// TIA Portal V18 export
// export: Created 2026-06-08T17:17:40.8310714Z, ExportSetting WithDefaults, DisplayName Totally Integrated Automation Portal, DisplayVersion V18, DisplayName TIA Portal Openness, DisplayVersion V18, DisplayName TIA Portal Version Control Interface, DisplayVersion V18, DisplayName STEP 7 Professional, DisplayVersion V18, DisplayName STEP 7 Safety, DisplayVersion V18, DisplayName WinCC Professional, DisplayVersion V18
ORGANIZATION_BLOCK "Main"   // OB1, LAD, ProgramCycle
TITLE = "Main Program Sweep (Cycle)"
{ S7_Optimized_Access := 'TRUE' }
VERSION : 0.1
// stored: AutoNumber true, IsIECCheckEnabled false, SetENOAutomatically false
BEGIN

REGION Network 1
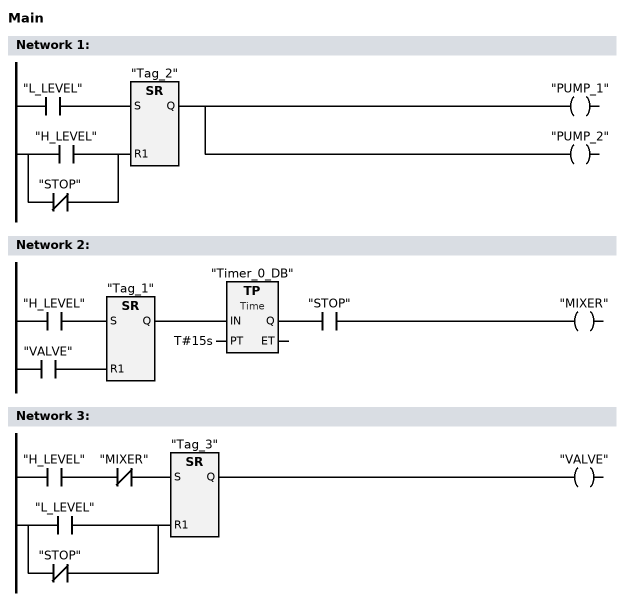
   RUNG wire#powerrail
      Contact( "L_LEVEL" )
      S_SR(operand := "Tag_2", r1 := wire#w1)
      wire#w2
      Coil( "PUMP_1" )
   END_RUNG
   RUNG wire#powerrail
      Contact( "H_LEVEL" )
   END_RUNG wire#w1
   RUNG wire#powerrail
      I_Contact( "STOP" )
   END_RUNG wire#w1
   RUNG wire#w2
      Coil( "PUMP_2" )
   END_RUNG
   // the same network as SCL:
   IF "L_LEVEL" THEN
       "Tag_2" := TRUE;   // SR flip-flop
   END_IF;
   IF "H_LEVEL" OR NOT "STOP" THEN "Tag_2" := FALSE; END_IF;
   "PUMP_1" := "Tag_2";
   "PUMP_2" := "Tag_2";
END_REGION

REGION Network 2
   RUNG wire#powerrail
      Contact( "H_LEVEL" )
      S_SR(operand := "Tag_1", r1 := wire#w1)
      { S7_Templates := "time_type := Time" } "Timer_0_DB".TP(pt := T#15s, et =>)
      Contact( "STOP" )
      Coil( "MIXER" )
   END_RUNG
   RUNG wire#powerrail
      Contact( "VALVE" )
   END_RUNG wire#w1
   // the same network as SCL:
   IF "H_LEVEL" THEN
       "Tag_1" := TRUE;   // SR flip-flop
   END_IF;
   IF "VALVE" THEN "Tag_1" := FALSE; END_IF;
   "Timer_0_DB".TP(IN := "Tag_1", PT := T#15s);
   "MIXER" := "Timer_0_DB".Q AND "STOP";
END_REGION

REGION Network 3
   RUNG wire#powerrail
      Contact( "H_LEVEL" )
      I_Contact( "MIXER" )
      S_SR(operand := "Tag_3", r1 := wire#w1)
      Coil( "VALVE" )
   END_RUNG
   RUNG wire#powerrail
      Contact( "L_LEVEL" )
   END_RUNG wire#w1
   RUNG wire#powerrail
      I_Contact( "STOP" )
   END_RUNG wire#w1
   // the same network as SCL:
   IF "H_LEVEL" AND NOT "MIXER" THEN
       "Tag_3" := TRUE;   // SR flip-flop
   END_IF;
   IF "L_LEVEL" OR NOT "STOP" THEN "Tag_3" := FALSE; END_IF;
   "VALVE" := "Tag_3";
END_REGION
END_ORGANIZATION_BLOCK
